// Mitsubishi GX Works2 project: InterLock   PLC: Q03UDV

PROGRAM MAIN
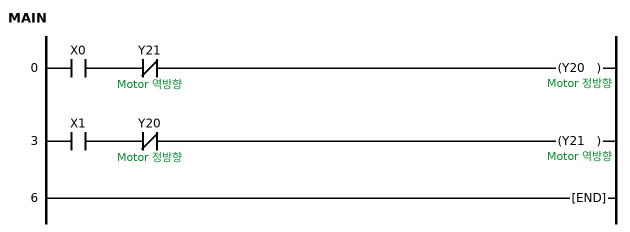
0     LD      X0
      ANI     Y21  ; Motor 역방향
      OUT     Y20  ; Motor 정방향
3     LD      X1
      ANI     Y20  ; Motor 정방향
      OUT     Y21  ; Motor 역방향
6     END
END_PROGRAM
